{attribute 'qualified_only'}
{attribute 'strict'}
TYPE EReportType_t :
(
	eUnitTestReport := 0,
	eExternalReport
);
END_TYPE

(* stored: Version 1.1.0.1, ProductVersion 3.1.4024.9
   DUT EReportType_t: Id {d6fbd902-e500-4190-ba1b-36716e3ffec5} *)
